{attribute 'linkalways'} 
{attribute 'no_explicit_call' := 'This FB is a CLASS and must be accessed using methods or properties'}
{attribute 'enable_dynamic_creation'}
FUNCTION_BLOCK _ETcVnEdgeDirection EXTENDS EnumDatatypeBase
VAR
	localData : ETcVnEdgeDirection;
	activeData : REFERENCE TO ETcVnEdgeDirection;
	enumBaseDatatype : _DINT(localData);
END_VAR

METHOD PRIVATE AddLocalEnumeration
VAR_INPUT
	Enumeration : T_MAXSTRING;
	Value : ETcVnEdgeDirection;
END_VAR
AddEnumeration(Enumeration, Value);
END_METHOD

PROPERTY PUBLIC Address : PVOID
GET
Address := ADR(activeData);
END_GET
END_PROPERTY

METHOD PUBLIC ClearReference
VAR_INPUT
END_VAR
activeData REF= localData;
SetBaseDatatypeReference();
END_METHOD

METHOD PUBLIC Clone : I_Datatype
VAR
    pClone : POINTER TO _ETcVnEdgeDirection;
END_VAR
pClone := __NEW(_ETcVnEdgeDirection(InitialValue := Value));
Clone := pClone^;
END_METHOD

METHOD FB_init : BOOL
VAR_INPUT
	bInitRetains : BOOL; // if TRUE, the retain variables are initialized (warm start / cold start)
	bInCopyCode : BOOL;  // if TRUE, the instance afterwards gets moved into the copy code (online change)
	InitialValue : ETcVnEdgeDirection;
END_VAR
localData := InitialValue;
AddBaseDatatype(enumBaseDatatype);
ClearReference();

AddLocalEnumeration('TCVN_ED_DARK_TO_LIGHT', ETcVnEdgeDirection.TCVN_ED_DARK_TO_LIGHT);
AddLocalEnumeration('TCVN_ED_LIGHT_TO_DARK', ETcVnEdgeDirection.TCVN_ED_LIGHT_TO_DARK);
END_METHOD

PROPERTY PUBLIC Identifier : T_MAXSTRING
GET
Identifier := 'ETcVnEdgeDirection';
END_GET
END_PROPERTY

METHOD IsEnumeratorValueEqual : BOOL
VAR_INPUT
	Enumerator : I_KeyValueForwardEnumerator;
END_VAR
VAR
	storedValue : ETcVnEdgeDirection;
END_VAR
IF NOT Enumerator.TryGet(storedValue) THEN
	RETURN;
END_IF

IsEnumeratorValueEqual := storedValue = activeData;
END_METHOD

METHOD PUBLIC MakeReferenceTo
VAR_INPUT
	ReferenceTarget : REFERENCE TO ETcVnEdgeDirection;
END_VAR
activeData REF= ReferenceTarget;
SetBaseDatatypeReference();
END_METHOD

METHOD PROTECTED SetBaseDatatypeReference
VAR_INPUT
END_VAR
enumBaseDatatype.MakeReferenceTo(activeData);
END_METHOD

PROPERTY PUBLIC Size : UDINT
GET
Size := SIZEOF(activeData);
END_GET
END_PROPERTY

METHOD TryMakeReferenceTo : BOOL
VAR_INPUT
	Target : I_Datatype;
END_VAR
VAR
	targetAsEnum : I_EnumDatatype;
	pTargetData : POINTER TO ETcVnEdgeDirection;
END_VAR
IF NOT Target.TryResolveAsEnumDatatype(targetAsEnum) THEN
	RETURN;
END_IF

IF targetAsEnum.Identifier <> Identifier THEN
	RETURN;
END_IF

pTargetData := Target.Address;
activeData REF= pTargetData^;
SetBaseDatatypeReference();
TryMakeReferenceTo := TRUE;
END_METHOD

PROPERTY PUBLIC Value : ETcVnEdgeDirection
GET
Value := activeData;
END_GET
SET
activeData := Value;
END_SET
END_PROPERTY

END_FUNCTION_BLOCK

(* stored: Version 1.1.0.1, ProductVersion 3.1.4024.12
   POU _ETcVnEdgeDirection: Id {aef29b18-f0fa-4fe3-a666-440918ee6082}, SpecialFunc None
   Folder Constructor: Id {317391ae-ecee-4ca6-8296-502d451dc175}
   Folder Private: Id {a1f929d2-18e7-472b-853a-fdd7124b98df}
   Folder Protected: Id {40e906be-d402-4bf5-96e4-4c9cff7835f9}
   Method AddLocalEnumeration: Id {6e776ac0-eb33-4a97-8d8f-0bb6f5a20818}
   Property Address: Id {a9118142-90c3-4a1e-9bad-5b2cc7d77c76}
   Get Get: Id {980c9d53-b664-4f12-b03b-d24ac06298b5}
   Method ClearReference: Id {4f47e37d-fa6c-4a69-8947-a5e9e3f697af}
   Method Clone: Id {7c61cbe0-19a9-4fb9-a2c3-0abba6273950}
   Method FB_init: Id {86bff729-b259-42b3-9d4c-2a8188d55c05}
   Property Identifier: Id {72b382a5-5211-4efb-a679-f7711b720db4}
   Get Get: Id {dedb510d-b4e8-4d0e-a873-b4400793b4dd}
   Method IsEnumeratorValueEqual: Id {ceac6ad5-e19c-4c2b-9611-9994ff7cc74f}
   Method MakeReferenceTo: Id {a5df675c-d48c-4b0d-80fa-c0f83b160015}
   Method SetBaseDatatypeReference: Id {4882ed8a-aecc-4d66-a166-51887a9e9deb}
   Property Size: Id {444ac385-fbf5-491b-869f-af6c31c0c013}
   Get Get: Id {a121b5e2-aac6-406c-99e5-41008cd787f7}
   Method TryMakeReferenceTo: Id {e67a1eb4-c725-4def-a7ae-c5740732713b}
   Property Value: Id {9fe44db3-88f4-4ad8-b292-cd2e4fdd68b3}
   Get Get: Id {9b40b029-f42a-4bc5-81fb-3885986df913}
   Set Set: Id {c18177c0-b447-49e7-bb6c-be70ed9a44f7} *)
